(* FB_Cylinder		- number of control signals:
							one direction is controllable
					- type of feedback:
							feedback is base and work position
*)

FUNCTION_BLOCK FB_CylinderBase IMPLEMENTS I_Cylinder
VAR_INPUT
	bAtBasePos		AT %I*		:	BOOL;		// Hardware input signal: cylinder is at base position
	bAtWorkPos		AT %I*		:	BOOL;		// Hardware input signal: cylinder is at work position
END_VAR
VAR_OUTPUT
	bMoveToWork		AT %Q*		:	BOOL;		// Hardware output signal to move cylinder to work position
END_VAR
VAR
END_VAR

// =================================================
;
// =================================================

{warning 'add property implementation'}
PROPERTY bState_AtBasePos : BOOL
GET
bState_AtBasePos := THIS^.bAtBasePos;
END_GET
END_PROPERTY

{warning 'add property implementation'}
PROPERTY bState_AtWorkPos : BOOL
GET
bState_AtWorkPos := THIS^.bAtWorkPos;
END_GET
END_PROPERTY

{warning 'add property implementation'}
PROPERTY bState_MoveToWork : BOOL
GET
bState_MoveToWork := THIS^.bMoveToWork;
END_GET
END_PROPERTY

METHOD MoveToBase
StateMachine(	bBasePosReq		:=		TRUE,
				bWorkPosReq		:=		FALSE);
END_METHOD

METHOD MoveToWork
StateMachine(	bBasePosReq		:=		FALSE,
				bWorkPosReq		:=		TRUE);
END_METHOD

METHOD Reset
THIS^.bMoveToWork		:=		FALSE;
END_METHOD

METHOD PROTECTED StateMachine
VAR_INPUT
	bBasePosReq		:	BOOL;
	bWorkPosReq		:	BOOL;
END_VAR
IF bWorkPosReq THEN
	THIS^.bMoveToWork 	:=		TRUE;
END_IF

IF bBasePosReq OR NOT bWorkPosReq THEN
	THIS^.bMoveToWork	:=		FALSE;
END_IF
END_METHOD

END_FUNCTION_BLOCK

(* stored: Version 1.1.0.1, ProductVersion 3.1.4024.15
   POU FB_CylinderBase: Id {06a0551f-8b6e-453f-a160-073165307183}, SpecialFunc None
   Property bState_AtBasePos: Id {881e8349-fc70-4146-ac9d-ea0f415c5c5a}
   Get Get: Id {5340a569-6d42-4fb1-b3c0-5dc7eb099938}
   Property bState_AtWorkPos: Id {8f2fdb38-3da8-4d15-b7bf-86f29da61513}
   Get Get: Id {55f81513-f914-4fa1-9596-85260b9daf6a}
   Property bState_MoveToWork: Id {a3d727ab-d38d-4baa-a490-84c48c40ab31}
   Get Get: Id {3a477c21-ff94-4ae8-9cf2-5049ade9e341}
   Method MoveToBase: Id {aaeca242-64eb-4206-b0a0-646874e50979}
   Method MoveToWork: Id {2e0e39fe-2f23-4963-a258-600a5f9f7a0b}
   Method Reset: Id {07b8644e-50b9-4ec4-8155-915c20b2e1bd}
   Method StateMachine: Id {7558132b-b58b-4df3-a067-5a584208c9d2} *)
